TYPE ST_Chamber1SingleProcessStageTimeConfigs :
STRUCT
	Prepare : ST_Chamber1SingleProcessStageTimeConfig;
	LiftReady : ST_Chamber1SingleProcessStageTimeConfig;
	SpinAlign : ST_Chamber1SingleProcessStageTimeConfig;
	ConcurrentProcessEntry : ST_Chamber1SingleProcessStageTimeConfig;
	SpinRampUp : ST_Chamber1SingleProcessStageTimeConfig;
	ProcessHold : ST_Chamber1SingleProcessStageTimeConfig;
	ConcurrentProcessExit : ST_Chamber1SingleProcessStageTimeConfig;
	SpinStandby : ST_Chamber1SingleProcessStageTimeConfig;
END_STRUCT
END_TYPE

(* stored: Version 1.1.0.1, ProductVersion 3.1.4026.18
   DUT ST_Chamber1SingleProcessStageTimeConfigs: Id {5252657b-d113-4ec3-8605-d510db42a751} *)
